FUNCTION_BLOCK FB_Room
VAR_INPUT
END_VAR
VAR_OUTPUT
END_VAR
VAR
	_aLamps		: ARRAY [1..10] OF FB_Lamp;
END_VAR

METHOD CalcPowerConsumption : UDINT
VAR_INPUT
END_VAR
VAR
	nLamp		:	INT;
END_VAR
FOR nLamp := 1 TO 10 DO
	CalcPowerConsumption := CalcPowerConsumption + refLamps[nLamp].nPowerConsumption;
END_FOR
END_METHOD

PROPERTY refLamps : REFERENCE TO ARRAY [1..10] OF FB_Lamp
GET
refLamps REF= THIS^._aLamps;
END_GET
END_PROPERTY

END_FUNCTION_BLOCK

(* stored: Version 1.1.0.1, ProductVersion 3.1.4024.12
   POU FB_Room: Id {7fb42700-b5b2-49df-a16f-73b5771ffe74}, SpecialFunc None
   Method CalcPowerConsumption: Id {b74f6046-ee06-4390-8760-063250eb3c33}
   Property refLamps: Id {6f5673cc-7bb1-4b5f-801c-3bfac429d442}
   Get Get: Id {3558468f-ea6a-486d-b0e1-4e3d93742db7} *)
